// TIA Portal V17 export
// export: Created 2023-04-20T09:49:48.3040453Z, ExportSetting WithDefaults, DisplayName Totally Integrated Automation Portal, DisplayVersion V17, DisplayName TIA Portal Openness, DisplayVersion V17, DisplayName TIA Portal Version Control Interface, DisplayVersion V17, DisplayName STEP 7 Professional, DisplayVersion V17, DisplayName STEP 7 Safety, DisplayVersion V17, DisplayName WinCC Advanced, DisplayVersion V17
VAR_GLOBAL   // PLC tag table "IO"
   IB_0 AT %IB0 : Byte;
   IB_1 AT %IB1 : Byte;
   QB_0 AT %QB0 : Byte;
   QB_1 AT %QB1 : Byte;
END_VAR
